# EPICS alarm handler configuration: mps_database/bareTest/alarms/areas/mpln_unds_mp05.alhConfig
GROUP NULL MPLN:UNDS:MP05:1
$ALIAS MPS Link Node 213
$GUIDANCE
LTUH MPS
   Group Name: MPLN:UNDS:MP05:1
   Summary PV:  MPLN:UNDS:MP05:1:STATSUMY
$END
CHANNEL  MPLN:UNDS:MP05:1    MPLN:UNDS:MP05:1:MPS_EN_RBV		-----
CHANNEL  MPLN:UNDS:MP05:1    MPLN:UNDS:MP05:1:LC1_MODE_RBV		-----
